FUNCTION LogMessage : DINT
VAR_INPUT
	msg		: STRING;
	hSocket	: T_HSOCKET;
END_VAR
VAR
END_VAR

IF GVL_TCP.G_bLogDebugMessages THEN
	LogMessage := ADSLOGDINT( ADSLOG_MSGTYPE_HINT OR ADSLOG_MSGTYPE_LOG, CONCAT( msg, ' :handle: %d' ), UDINT_TO_DINT(hSocket.handle)  );
ELSE
	LogMessage := 0;
END_IF

END_FUNCTION

(* stored: Version 1.1.0.1, ProductVersion 3.1.4024.3
   POU LogMessage: Id {cf020442-2fc1-4f73-8ea9-87a0ac6ae13e}, SpecialFunc None *)
